TYPE ST_System_Ampel_Steuerung :
STRUCT
	Regelung_Sollw		: ST_Steuerung_auto_manu_opti_AMPELSIGNAL;
END_STRUCT
END_TYPE

(* stored: Version 1.1.0.1, ProductVersion 3.1.4024.9
   DUT ST_System_Ampel_Steuerung: Id {b91e71d4-ce32-4a8b-98d1-4be5d0841d0d} *)
